FUNCTION_BLOCK Faults6
VAR_INPUT
END_VAR
VAR_OUTPUT
END_VAR
VAR
END_VAR

END_FUNCTION_BLOCK

(* stored: Version 1.1.0.1, ProductVersion 3.1.4024.11
   POU Faults6: Id {19469f92-2967-441c-8541-f1bae9feeb43}, SpecialFunc None *)
